TYPE ST_MC_Status :
STRUCT
	
	Status		: BOOL;
	Done		: BOOL;
	Busy		: BOOL;
	Error		: BOOL;
	Active		: BOOL;
	CmdAborted	: BOOL;
	InVelocity	: BOOL;
	ErrorID		: UDINt;
	
END_STRUCT
END_TYPE

(* stored: Version 1.1.0.1, ProductVersion 3.1.4024.10
   DUT ST_MC_Status: Id {be86b6f6-eafd-45aa-aeba-8cf3a68a4205} *)
